TYPE ST_Event :
STRUCT
	eEventType :E_EventType;
	eEventSeverity: Tc3_EventLogger.TcEventSeverity;
	nEventIdentity: UDINT;
	sEventText: STRING(255);
	dtTimestamp: DATE_AND_TIME;
END_STRUCT
END_TYPE

(* stored: Version 1.1.0.1, ProductVersion 3.1.4024.12
   DUT ST_Event: Id {939161b6-c637-4bad-9bc5-d3aea15b9aec} *)
